{attribute addProperty BoxType "EL3632-0000-0022"}
{attribute addProperty Id "STATUSAT %I*STATUS_84521898162"}
{attribute addProperty CRC "3729672571"}
{attribute addProperty SizeInBites "16"}
{attribute addProperty SizeInBytes "2"}
TYPE Ch1_Status_DE4E497B :
STRUCT
	{attribute addProperty Name "STATUS"}
	STATUS AT %I* : STATUS_84521898;
END_STRUCT
END_TYPE

(* stored: Version 1.2.0.0, ProductVersion 3.1.4024.9
   DUT Ch1_Status_DE4E497B: Id {d862920c-4ef5-4b7f-8cca-1d84e0b654c5} *)
